//==================================================================================================
//								RJM Maszyny sp. z o.o.
//									22.06.2022
//	Obsługa przycisku ze stykiem NC
// 	v1.0	|| TC v 3.1.4024.22		|| - pierwsza wersja
//==================================================================================================
FUNCTION_BLOCK FB_Przycisk_NC IMPLEMENTS ITF_Przycisk
VAR
	bStyk							AT %I*	: BOOL;
	bPodswietlenie					AT %Q*	: BOOL;
END_VAR

PROPERTY CzyNacisniety : BOOL
GET
CzyNacisniety								:= NOT bStyk;
END_GET
END_PROPERTY

PROPERTY Podswietlenie : BOOL
SET
bPodswietlenie								:= Podswietlenie;
END_SET
END_PROPERTY

END_FUNCTION_BLOCK

(* stored: Version 1.1.0.1, ProductVersion 3.1.4024.11
   POU FB_Przycisk_NC: Id {6319c024-154b-46d0-90c3-ab1a7fbadabd}, SpecialFunc None
   Property CzyNacisniety: Id {c8e99589-ae89-49ad-a359-5ca4e4ae6fba}
   Get Get: Id {1cd11f39-c7d1-4f37-bf68-2e26ade25f76}
   Property Podswietlenie: Id {5a7b5426-5f86-4062-8d50-8d094f90f338}
   Set Set: Id {7440f10a-6156-439e-978b-c17324af39b9} *)
